PROGRAM MAIN
VAR
END_VAR

DatabasePyAds();

END_PROGRAM

(* stored: Version 1.1.0.1, ProductVersion 3.1.4024.2
   POU MAIN: Id {681a437c-8c84-41fd-92aa-e39d4e2b0600}, SpecialFunc None *)
